SUBAPPLICATION Uebung_010e2 (* SR und T-Flip-Flop mit 3x SoftKey (Softkey_IE, SK_RELEASED) mit GreenWhiteBackground am Toggle-SoftKey mit Subapp *)
  (* Standard: 61499-2; Description: Copyright (c) 2026 Meisterschulen am Ostbahnhof This program and the accompanying materials are made available under the terms of the Eclipse Public License 2.0 which is available at https://www.eclipse.org/legal/epl-2.0/ SPDX-License-Identifier: EPL-2.0 *)
  (* Version 1.0, 2026-09-02, Franz Höpfinger, Meisterschulen am Ostbahnhof, initial API and implementation and/or initial documentation *)
  PACKAGE Uebungen;
  IMPORT Uebungen::const::UT::DefaultPool::SoftKey_F1;
  IMPORT Uebungen::const::UT::DefaultPool::SoftKey_F2;
  IMPORT Uebungen::const::UT::DefaultPool::SoftKey_F3;
  IMPORT logiBUS::io::DQ::logiBUS_DO::Output_Q1;
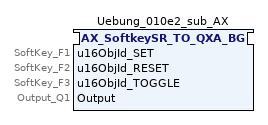
  SUBAPPS
    Uebung_010e2_sub_AX : MyLib::sys::AX_SoftkeySR_TO_QXA_BG(u16ObjId_SET := SoftKey_F1 (* Object ID SET SoftKey *), u16ObjId_RESET := SoftKey_F2 (* Object ID RESET SoftKey *), u16ObjId_TOGGLE := SoftKey_F3 (* Object ID TOGGLE SoftKey (auch fuer GreenWhiteBackground) *), Output := Output_Q1 (* Identify the Output Output_Q1..Q8 *));
  END_SUBAPPS
END_SUBAPPLICATION
